# EPICS alarm handler configuration: epics/epics_alh/alarms_list_BeamDAQ.alhConfig
GROUP NULL BeamDAQ
